// TIA Portal V15.1 export
// export: Created 2024-06-21T08:40:57.6277466Z, ExportSetting WithDefaults, DisplayName Totally Integrated Automation Portal, DisplayVersion V15.1 Update 5, DisplayName TIA Portal Openness, DisplayVersion V15.1 Update 5, DisplayName SINAMICS Startdrive Advanced, DisplayVersion V15.1, DisplayName G130, G150, S120, S150, SINAMICS MV, S210, DisplayVersion V15.1, DisplayName G110M, G120, G120C, G120D, G120P, DisplayVersion V15.1, DisplayName STEP 7 Professional, DisplayVersion V15.1 Update 5, DisplayName STEP 7 Safety, DisplayVersion V15.1, DisplayName WinCC Professional, DisplayVersion V15.1 Update 5, DisplayName SIMATIC Visualization Architect, DisplayVersion V15.1
FUNCTION_BLOCK "L1SafetyCh1Alarm"   // FB1421, FBD
TITLE = L1SafetyCh1Alarm
{ S7_Optimized_Access := 'FALSE' }
AUTHOR : VCC
FAMILY : AlarmHnd
NAME : 1SafeAlm
VERSION : 0.1
// ================================================================================
// This module is used everywhere one alarm shall be generated when one security 
// input becomes False.
// The alarm can be True only when the input Enable Alarm is also True.
// When the condition to generate the alarm is not fullfilled, a boolean output is 
// available to inform the upper level that the alarm can be reset.
// The alarm is reset by means of the AlarmResetPB signal.
// 
// This module generates also a word containing all necessary information for HMI 
// Icon animation, and a word with all information for HMI safety module 
// diagnostic 
// screen. 
// ================================================================================
// stored: AutoNumber false, IsIECCheckEnabled false, SetENOAutomatically False, UDAEnableTagReadback false
   VAR_INPUT
      I_Input { ExternalAccessible := 'False'; ExternalVisible := 'False'; ExternalWritable := 'False'} : Bool;   // Input safety alarm (normally closed)
      I_AlarmClass { ExternalAccessible := 'False'; ExternalVisible := 'False'; ExternalWritable := 'False'} : Char;   // Alarm class -> A - B - C - D or E
      I_EnableAlarm { ExternalAccessible := 'False'; ExternalVisible := 'False'; ExternalWritable := 'False'} : Bool := TRUE;   // Enable alarm from upper level (0=disable/1=enable)
      I_AlarmResetPB { ExternalAccessible := 'False'; ExternalVisible := 'False'; ExternalWritable := 'False'} : Bool;   // Alarm reset pushbutton is activated
      I_SafetyCard_PASS_OUT { ExternalAccessible := 'False'; ExternalVisible := 'False'; ExternalWritable := 'False'} : Bool;   // Automatically generated DB from F-Modul (F-Peripherie DB)
      I_SafetyCard_ACK_REQ { ExternalAccessible := 'False'; ExternalVisible := 'False'; ExternalWritable := 'False'} : Bool;   // Automatically generated DB from F-Modul (F-Peripherie DB)
      I_SafetyCard_DIAG { ExternalAccessible := 'False'; ExternalVisible := 'False'; ExternalWritable := 'False'} : Byte;   // Automatically generated DB from F-Modul (F-Peripherie DB)
      I_SafetyCardHWSub { ExternalAccessible := 'False'; ExternalVisible := 'False'; ExternalWritable := 'False'} : HW_SUBMODULE;   // Safety I/O connection hardware
      I_ChannelNr { ExternalAccessible := 'False'; ExternalVisible := 'False'; ExternalWritable := 'False'} : Int;   // Used Channel Nr (Value : 0 - 7)
   END_VAR
   VAR_OUTPUT
      O_Alarm { ExternalAccessible := 'False'; ExternalVisible := 'False'; ExternalWritable := 'False'} : Bool;   // Alarm
      O_AlarmABCondition { ExternalAccessible := 'False'; ExternalVisible := 'False'; ExternalWritable := 'False'} : Bool;   // Alarm AB condition
      H_IAnim { ExternalAccessible := 'False'; ExternalVisible := 'False'; ExternalWritable := 'False'} : Word;   // Icon Animation
   END_VAR
   VAR DB_SPECIFIC
      H_Out : Struct   // HMI
         Anim : Word;   // HMI Animation of the object
         DBnr : Int;   // HMI Animation DB number
      END_STRUCT;
      Alarm { ExternalAccessible := 'False'; ExternalVisible := 'False'; ExternalWritable := 'False'} : Bool;   // Alarm
      AlarmClass_A { ExternalAccessible := 'False'; ExternalVisible := 'False'; ExternalWritable := 'False'} : Bool;   // The alarm is from alarm class A
      AlarmClass_B { ExternalAccessible := 'False'; ExternalVisible := 'False'; ExternalWritable := 'False'} : Bool;   // The alarm is from alarm class B
      AlarmClass_C { ExternalAccessible := 'False'; ExternalVisible := 'False'; ExternalWritable := 'False'} : Bool;   // The alarm is from alarm class C
      AlarmClass_D { ExternalAccessible := 'False'; ExternalVisible := 'False'; ExternalWritable := 'False'} : Bool;   // The alarm is from alarm class D
      QbadCh1 { ExternalAccessible := 'False'; ExternalVisible := 'False'; ExternalWritable := 'False'} : Bool;   // Passivation first Channel
      Ack_Req { ExternalAccessible := 'False'; ExternalVisible := 'False'; ExternalWritable := 'False'} : Bool;   // Acknowledgement request
      Timeout_F_I_O { ExternalAccessible := 'False'; ExternalVisible := 'False'; ExternalWritable := 'False'} : Bool;   // Timeout detected by F-I/O
      ChannelFault_F_I_O { ExternalAccessible := 'False'; ExternalVisible := 'False'; ExternalWritable := 'False'} : Bool;   // F-I/O fault or channel fault detected by F-I/O
      CRCSeqError_F_I_O { ExternalAccessible := 'False'; ExternalVisible := 'False'; ExternalWritable := 'False'} : Bool;   // CRC error or sequence number error detected by F-I/O
      Timeout_F_Sys { ExternalAccessible := 'False'; ExternalVisible := 'False'; ExternalWritable := 'False'} : Bool;   // Timeout detected by F-System
      SeqError_F_Sys { ExternalAccessible := 'False'; ExternalVisible := 'False'; ExternalWritable := 'False'} : Bool;   // Sequence number error detected by F-system
      CRCError_F_Sys { ExternalAccessible := 'False'; ExternalVisible := 'False'; ExternalWritable := 'False'} : Bool;   // CRC error detected by F-system
      AlarmCond { ExternalAccessible := 'False'; ExternalVisible := 'False'; ExternalWritable := 'False'} : Bool;   // Alarm condition
      RetValueData { ExternalAccessible := 'False'; ExternalVisible := 'False'; ExternalWritable := 'False'} : Int;   // Status variable (SFC14)
      DBnr { ExternalAccessible := 'False'; ExternalVisible := 'False'; ExternalWritable := 'False'} : Int;   // HMI DB number
   END_VAR
   VAR_TEMP
      T_DataFromSafetyCard : Struct   // Temp structure : receive data's from Safety Card
         Byte0_Bit0_Spare : Bool;
         Byte0_Bit1_Spare : Bool;
         Byte0_Bit2_Spare : Bool;
         Byte0_Bit3_Spare : Bool;
         Byte0_Bit4_Spare : Bool;
         Byte0_Bit5_Spare : Bool;
         Byte0_Bit6_Spare : Bool;
         Byte0_Bit7_Spare : Bool;
         Byte1_Bit0_QBadCh0 : Bool;
         Byte1_Bit1_QBadCh1 : Bool;
         Byte1_Bit2_QBadCh2 : Bool;
         Byte1_Bit3_QBadCh3 : Bool;
         Byte1_Bit4_QBadCh4 : Bool;
         Byte1_Bit5_QBadCh5 : Bool;
         Byte1_Bit6_QBadCh6 : Bool;
         Byte1_Bit7_QBadCh7 : Bool;
         Byte2_bit0_Spare : Bool;
         Byte2_bit1_Spare : Bool;
         Byte2_bit2_Spare : Bool;
         Byte2_bit3_Spare : Bool;
         Byte2_bit4_Spare : Bool;
         Byte2_bit5_Spare : Bool;
         Byte2_bit6_Spare : Bool;
         Byte2_bit7_Spare : Bool;
         Byte3_Bit0_Spare : Bool;
         Byte3_Bit1_Spare : Bool;
         Byte3_Bit2_Spare : Bool;
         Byte3_Bit3_Spare : Bool;
         Byte3_Bit4_Spare : Bool;
         Byte3_Bit5_Spare : Bool;
         Byte3_Bit6_Spare : Bool;
         Byte3_Bit7_Spare : Bool;
         Byte4_bit0_Spare : Bool;
         Byte4_bit1_Spare : Bool;
         Byte4_bit2_Spare : Bool;
         Byte4_bit3_Spare : Bool;
         Byte4_bit4_Spare : Bool;
         Byte4_bit5_Spare : Bool;
         Byte4_bit6_Spare : Bool;
         Byte4_bit7_Spare : Bool;
         Byte5_bit0_Spare : Bool;
         Byte5_bit1_Spare : Bool;
         Byte5_bit2_Spare : Bool;
         Byte5_bit3_Spare : Bool;
         Byte5_bit4_Spare : Bool;
         Byte5_bit5_Spare : Bool;
         Byte5_bit6_Spare : Bool;
         Byte5_bit7_Spare : Bool;
      END_STRUCT;
   END_VAR
BEGIN

NETWORK
TITLE = **** 1 - Inputs **** DB number
// DB number
      L     DINO;
      T     #DBnr;

NETWORK
TITLE = **** 1 - Inputs **** Alarm class
// Alarm class
// Alarm class = D
      L     #I_AlarmClass;
      L     'D';
      ==I;
      =     #AlarmClass_D;

// Alarm class = C
      L     #I_AlarmClass;
      L     'C';
      ==I;
      =     #AlarmClass_C;

// Alarm class = B
      L     #I_AlarmClass;
      L     'B';
      ==I;
      =     #AlarmClass_B;

// Alarm class = A
      AN    #AlarmClass_B;
      AN    #AlarmClass_C;
      AN    #AlarmClass_D;
      =     #AlarmClass_A;


REGION Network 3: **** 1 - Inputs **** Safety I/O connection hardware
   // Safety I/O connection hardware
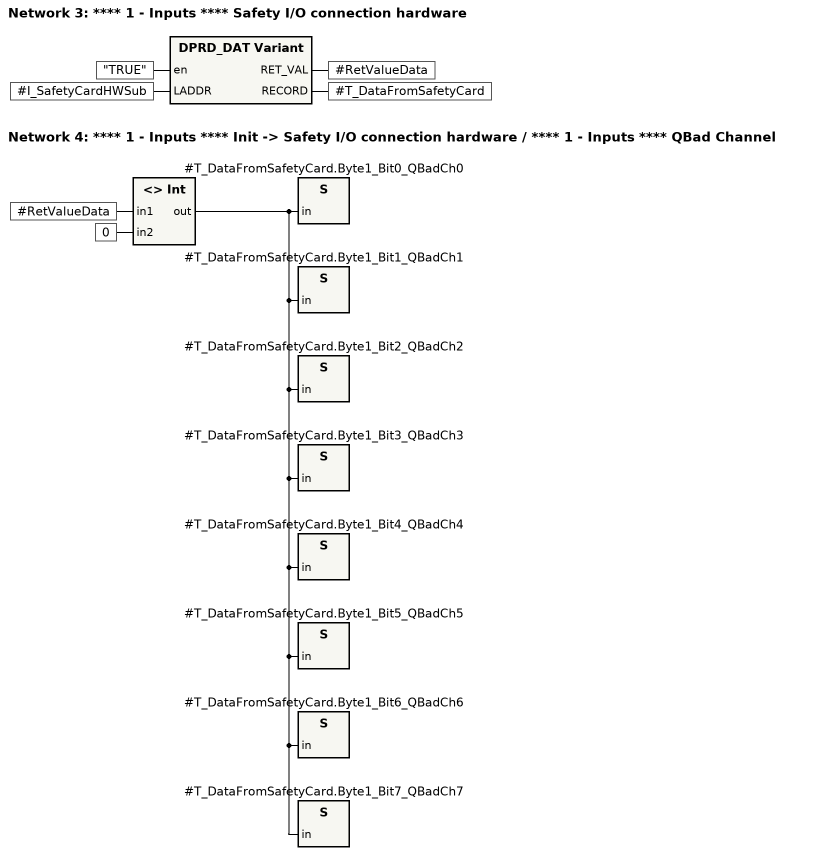
   IF "TRUE" THEN
       #RetValueData := DPRD_DAT(LADDR := #I_SafetyCardHWSub, RECORD => #T_DataFromSafetyCard);
   END_IF;
END_REGION

REGION Network 4: **** 1 - Inputs **** Init -> Safety I/O connection hardware / **** 1 - Inputs **** QBad Channel
   // Init -> Safety I/O connection hardware
   IF #RetValueData <> 0 THEN
       #T_DataFromSafetyCard.Byte1_Bit0_QBadCh0 := TRUE;
       #T_DataFromSafetyCard.Byte1_Bit1_QBadCh1 := TRUE;
       #T_DataFromSafetyCard.Byte1_Bit2_QBadCh2 := TRUE;
       #T_DataFromSafetyCard.Byte1_Bit3_QBadCh3 := TRUE;
       #T_DataFromSafetyCard.Byte1_Bit4_QBadCh4 := TRUE;
       #T_DataFromSafetyCard.Byte1_Bit5_QBadCh5 := TRUE;
       #T_DataFromSafetyCard.Byte1_Bit6_QBadCh6 := TRUE;
       #T_DataFromSafetyCard.Byte1_Bit7_QBadCh7 := TRUE;
   END_IF;
END_REGION

REGION Network 5: **** 1 - Inputs **** Qbad Channel 1
   // Qbad Channel 1
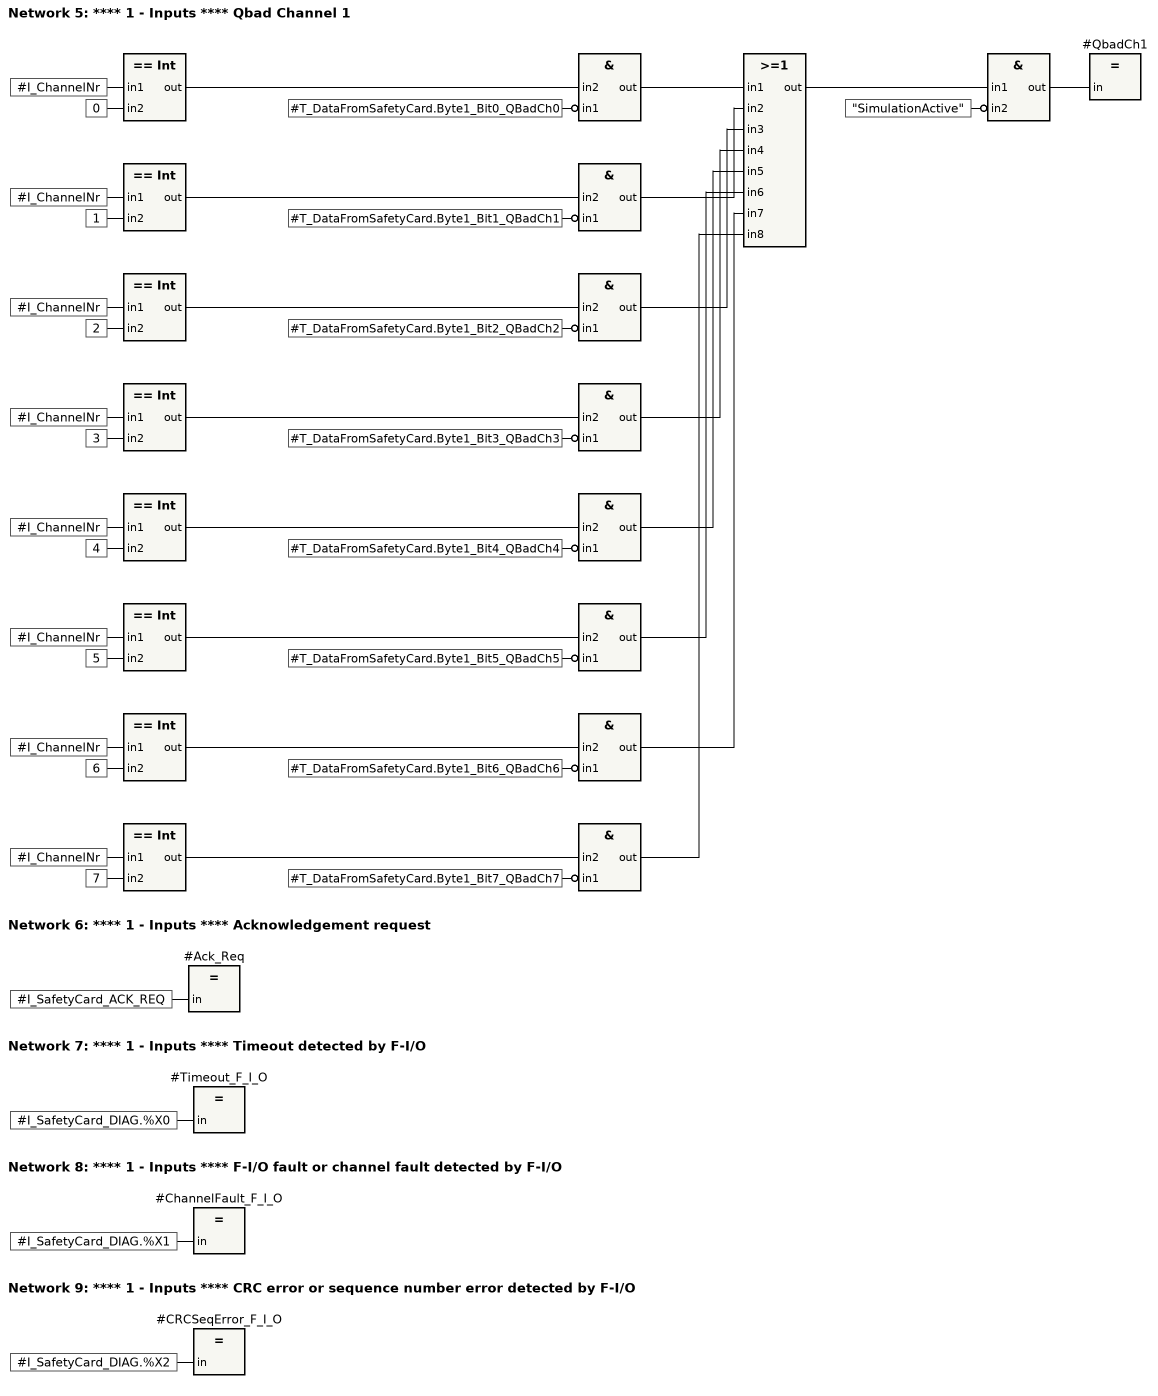
   #QbadCh1 := (((#I_ChannelNr = 0) AND NOT #T_DataFromSafetyCard.Byte1_Bit0_QBadCh0) OR ((#I_ChannelNr = 1) AND NOT #T_DataFromSafetyCard.Byte1_Bit1_QBadCh1) OR ((#I_ChannelNr = 2) AND NOT #T_DataFromSafetyCard.Byte1_Bit2_QBadCh2) OR ((#I_ChannelNr = 3) AND NOT #T_DataFromSafetyCard.Byte1_Bit3_QBadCh3) OR ((#I_ChannelNr = 4) AND NOT #T_DataFromSafetyCard.Byte1_Bit4_QBadCh4) OR ((#I_ChannelNr = 5) AND NOT #T_DataFromSafetyCard.Byte1_Bit5_QBadCh5) OR ((#I_ChannelNr = 6) AND NOT #T_DataFromSafetyCard.Byte1_Bit6_QBadCh6) OR ((#I_ChannelNr = 7) AND NOT #T_DataFromSafetyCard.Byte1_Bit7_QBadCh7)) AND NOT "SimulationActive";
END_REGION

REGION Network 6: **** 1 - Inputs **** Acknowledgement request
   // Acknowledgement request
   #Ack_Req := #I_SafetyCard_ACK_REQ;
END_REGION

REGION Network 7: **** 1 - Inputs **** Timeout detected by F-I/O
   // Timeout detected by F-I/O
   #Timeout_F_I_O := #I_SafetyCard_DIAG.%X0;
END_REGION

REGION Network 8: **** 1 - Inputs **** F-I/O fault or channel fault detected by F-I/O
   // F-I/O fault or channel fault detected by F-I/O
   #ChannelFault_F_I_O := #I_SafetyCard_DIAG.%X1;
END_REGION

REGION Network 9: **** 1 - Inputs **** CRC error or sequence number error detected by F-I/O
   // CRC error or sequence number error detected by F-I/O
   #CRCSeqError_F_I_O := #I_SafetyCard_DIAG.%X2;
END_REGION

REGION Network 10: **** 1 - Inputs **** Timeout detected by F-system
   // Timeout detected by F-system
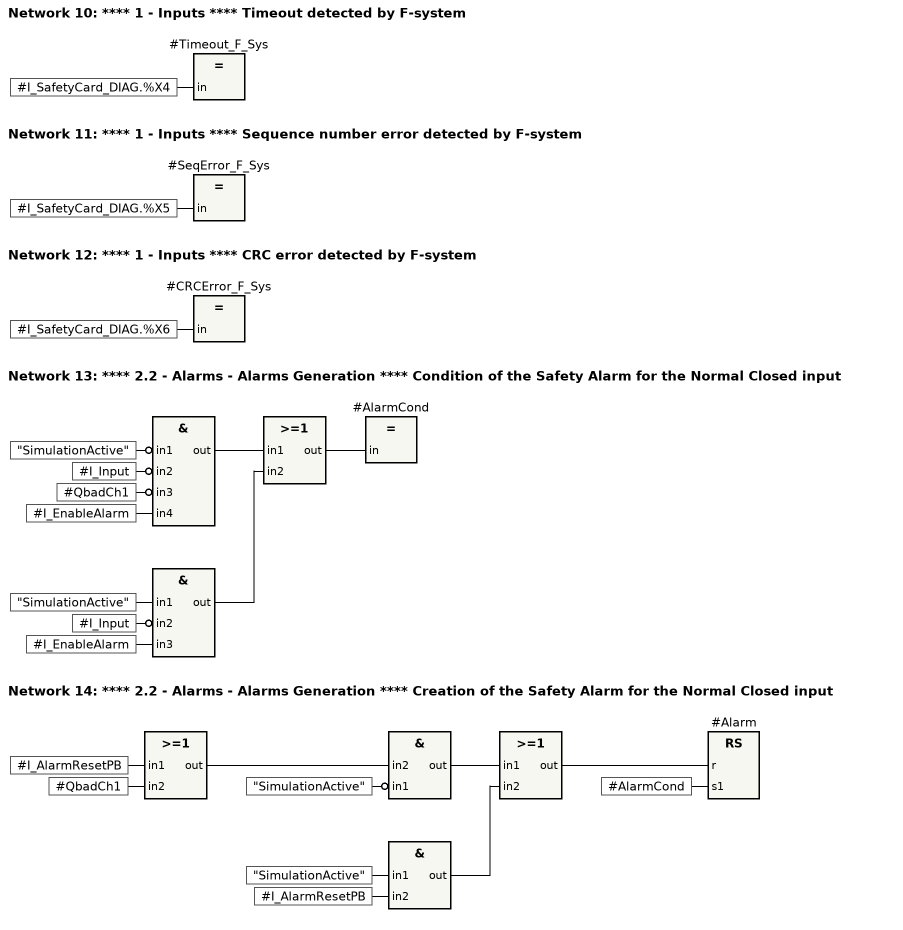
   #Timeout_F_Sys := #I_SafetyCard_DIAG.%X4;
END_REGION

REGION Network 11: **** 1 - Inputs **** Sequence number error detected by F-system
   // Sequence number error detected by F-system
   #SeqError_F_Sys := #I_SafetyCard_DIAG.%X5;
END_REGION

REGION Network 12: **** 1 - Inputs **** CRC error detected by F-system
   // CRC error detected by F-system
   #CRCError_F_Sys := #I_SafetyCard_DIAG.%X6;
END_REGION

REGION Network 13: **** 2.2 - Alarms - Alarms Generation **** Condition of the Safety Alarm for the Normal Closed input
   // Condition of the Safety Alarm for the Normal Closed input
   #AlarmCond := (NOT "SimulationActive" AND NOT #I_Input AND NOT #QbadCh1 AND #I_EnableAlarm) OR ("SimulationActive" AND NOT #I_Input AND #I_EnableAlarm);
END_REGION

REGION Network 14: **** 2.2 - Alarms - Alarms Generation **** Creation of the Safety Alarm for the Normal Closed input
   // Creation of the Safety Alarm for the Normal Closed input
   IF ((#I_AlarmResetPB OR #QbadCh1) AND NOT "SimulationActive") OR ("SimulationActive" AND #I_AlarmResetPB) THEN
       #Alarm := FALSE;   // RS flip-flop
   END_IF;
   IF #AlarmCond THEN #Alarm := TRUE; END_IF;
END_REGION

REGION Network 15: **** 4.6 - Mashine Status - Indications **** Icon Animation
   // Icon Animation
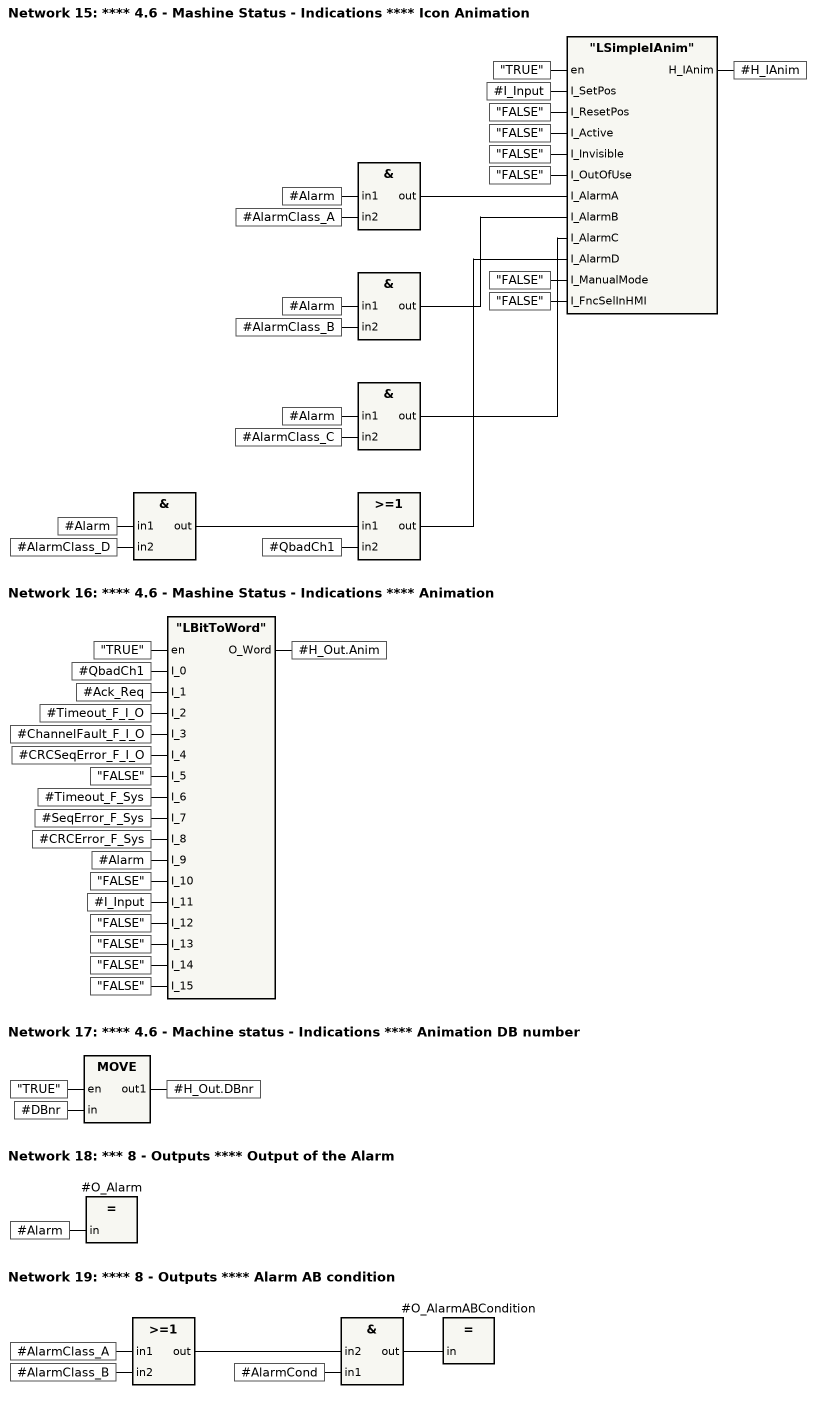
   IF "TRUE" THEN
       "LSimpleIAnim"(I_SetPos := #I_Input,
                      I_ResetPos := "FALSE",
                      I_Active := "FALSE",
                      I_Invisible := "FALSE",
                      I_OutOfUse := "FALSE",
                      I_AlarmA := #Alarm AND #AlarmClass_A,
                      I_AlarmB := #Alarm AND #AlarmClass_B,
                      I_AlarmC := #Alarm AND #AlarmClass_C,
                      I_AlarmD := (#Alarm AND #AlarmClass_D) OR #QbadCh1,
                      I_ManualMode := "FALSE",
                      I_FncSelInHMI := "FALSE",
                      H_IAnim => #H_IAnim);
   END_IF;
END_REGION

REGION Network 16: **** 4.6 - Mashine Status - Indications **** Animation
   // Animation
   IF "TRUE" THEN
       "LBitToWord"(I_0 := #QbadCh1,
                    I_1 := #Ack_Req,
                    I_2 := #Timeout_F_I_O,
                    I_3 := #ChannelFault_F_I_O,
                    I_4 := #CRCSeqError_F_I_O,
                    I_5 := "FALSE",
                    I_6 := #Timeout_F_Sys,
                    I_7 := #SeqError_F_Sys,
                    I_8 := #CRCError_F_Sys,
                    I_9 := #Alarm,
                    I_10 := "FALSE",
                    I_11 := #I_Input,
                    I_12 := "FALSE",
                    I_13 := "FALSE",
                    I_14 := "FALSE",
                    I_15 := "FALSE",
                    O_Word => #H_Out.Anim);
   END_IF;
END_REGION

REGION Network 17: **** 4.6 - Machine status - Indications **** Animation DB number
   // Animation DB number
   IF "TRUE" THEN #H_Out.DBnr := #DBnr; END_IF;
END_REGION

REGION Network 18: *** 8 - Outputs **** Output of the Alarm
   // Output of the Alarm
   #O_Alarm := #Alarm;
END_REGION

REGION Network 19: **** 8 - Outputs **** Alarm AB condition
   // Alarm AB condition
   #O_AlarmABCondition := (#AlarmClass_A OR #AlarmClass_B) AND #AlarmCond;
END_REGION
END_FUNCTION_BLOCK
